FUNCTION_BLOCK FB_Cylinder_DualPWM_DualTimer EXTENDS FB_Cylinder_NoSensor
VAR_INPUT
END_VAR
VAR_OUTPUT
END_VAR
VAR
	fbPWMControl		: FB_Enfield_LSV_PWM_SolenoidControl;
	
	//Internal Property Values
	nDutyCycle		: INT := 100;
	
END_VAR

PROPERTY DutyCycle : INT
GET
DutyCycle := nDutyCycle;
END_GET
SET
nDutyCycle := DutyCycle;
END_SET
END_PROPERTY

METHOD HardwareUpdate : BOOL
VAR_INPUT
END_VAR
SUPER^.HardwareUpdate();

IF bExtendCommand THEN
	fbPWMControl.Actuate(nDutyCycle);
ELSIF bRetractCommand THEN
	fbPWMControl.Actuate(nDutyCycle * -1);
ELSE
	fbPWMControl.Actuate(0);
END_IF
END_METHOD

END_FUNCTION_BLOCK

(* stored: Version 1.1.0.1, ProductVersion 3.1.4024.9
   POU FB_Cylinder_DualPWM_DualTimer: Id {bd0765f9-d5b5-41eb-b703-2e3258d3ef4c}, SpecialFunc None
   Folder 01_SUPER_Overrides: Id {86bd10f2-4685-4f68-bfaf-180b998b454c}
   Property DutyCycle: Id {2746359f-fb36-4e69-8211-8f6a3620eaf5}
   Get Get: Id {e4bc2f3b-cdd0-4d18-8858-256c10af0d95}
   Set Set: Id {d94aded6-354e-4ec6-afa1-1d48406a77c9}
   Method HardwareUpdate: Id {d7d74fec-42f1-4a65-95cb-b8d380a432fa} *)
